Yaskawa INFORM job: BUTT_WELD.JBI

/JOB
//NAME BUTT_WELD
//POS
///NPOS 9,0,0,0,0,0
///TOOL 5
///POSTYPE PULSE
///PULSE
C00000=-3,-50477,-58433,-6,-74934,492
C00001=-10903,50884,-493,-2391,-79024,-64715
C00002=-11058,51569,-1449,-2333,-77719,-64644
C00003=-6331,50752,-3005,-3989,-77266,-65791
C00004=-3955,50434,-3503,-4809,-77061,-66360
C00005=-1451,50248,-3859,-5656,-76848,-66964
C00006=-1343,50246,-3866,-5689,-76842,-66989
C00007=-1318,44844,3050,-5593,-85624,-67417
C00008=-3,-50477,-58433,-6,-74934,492
//INST
///DATE 2024/07/08 17:07
///ATTR SC,RW
///GROUP1 RB1
NOP
MOVJ C00000 VJ=4.00
MOVJ C00001 VJ=4.00
MOVL C00002 V=11.0
DOUT OT#(17) ON
ARCON AC=60 AVP=95
MOVL C00003 V=1.5
COMM ARCSET AC=60 AVP=115
COMM MOVL C00004 V=1.5
ARCSET AC=70 AVP=90
MOVL C00005 V=1.5
DOUT OT#(17) OFF
MOVL C00006 V=1.5
ARCOF
MOVJ C00007 VJ=2.00
MOVJ C00008 VJ=4.00
END
